// TIA Portal V19 program export: 1 tag tables, 0 data types, 0 data blocks, 5 code blocks (in call order from the OBs), 0 instance data blocks

VAR_GLOBAL   // PLC tag table "Default tag table"
   Stop_All AT %M0.0 : Bool;
   TestTag AT %M0.1 : Bool;
END_VAR

ORGANIZATION_BLOCK "Main"   // OB1, LAD, ProgramCycle
TITLE = "Main Program Sweep (Cycle)"
{ S7_Optimized_Access := 'TRUE' }
// h
// stored: SetENOAutomatically false
   VAR_INPUT
      Initial_Call : Bool;   // Initial call of this OB
      Remanence : Bool;   // =True, if remanent data are available
   END_VAR
   VAR_TEMP
      Start_All : Bool;
      ON : Bool;
   END_VAR
BEGIN

REGION Network 1
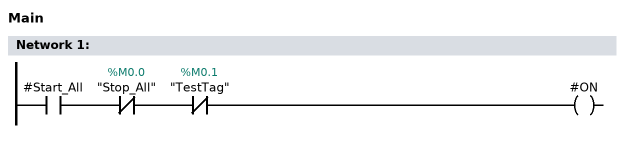
   RUNG wire#powerrail
      Contact( #Start_All )
      I_Contact( "Stop_All" )
      I_Contact( "TestTag" )
      Coil( #ON )
   END_RUNG
   // the same network as SCL:
   #ON := #Start_All AND NOT "Stop_All" AND NOT "TestTag";
END_REGION
END_ORGANIZATION_BLOCK

FUNCTION "NEW_FUNCTION" : Void   // FC2, LAD
TITLE = New Function Added
{ S7_Optimized_Access := 'TRUE' }
// stored: SetENOAutomatically false
BEGIN

REGION Network 1: New Function 1
   // Testing adding a new function.
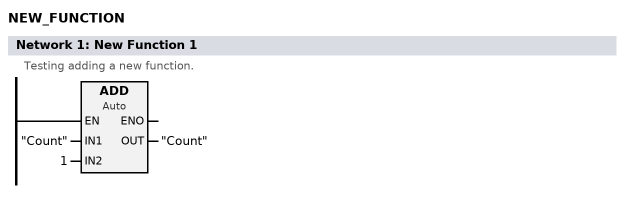
   RUNG wire#powerrail
      Add(in1 := "Count", in2 := 1, out => "Count")
   END_RUNG
   // the same network as SCL:
   "Count" := "Count" + 1;
END_REGION
END_FUNCTION

FUNCTION_BLOCK "SAMPLE_BLOCK"   // FB1, LAD
TITLE = Example Function Block - ie, Multiple Motors Start / Stop
{ S7_Optimized_Access := 'TRUE' }
// stored: MemoryReserve 100, SetENOAutomatically false
BEGIN

REGION Network 1: Drive 1 - Latching
   // Motor 1
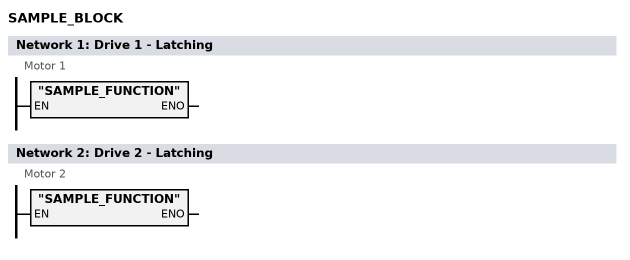
   RUNG wire#powerrail
      "SAMPLE_FUNCTION"()
   END_RUNG
   // the same network as SCL:
   "SAMPLE_FUNCTION"();
END_REGION

REGION Network 2: Drive 2 - Latching
   // Motor 2
   RUNG wire#powerrail
      "SAMPLE_FUNCTION"()
   END_RUNG
   // the same network as SCL:
   "SAMPLE_FUNCTION"();
END_REGION
END_FUNCTION_BLOCK

FUNCTION "SAMPLE_FUNCTION" : Void   // FC1, LAD
TITLE = SAMPLE FUNCTION FOR TESTING DOCUMENTATION
{ S7_Optimized_Access := 'TRUE' }
// stored: SetENOAutomatically false
   VAR_TEMP
      Start : Bool;   // Start Command
      Stop : Bool;   // Stop Command
      Running : Bool;   // Running ? (Y/N)
   END_VAR
BEGIN

REGION Network 1: Basic Latching Function
   // This is A Comment to Test The Documentation Prints Correctly
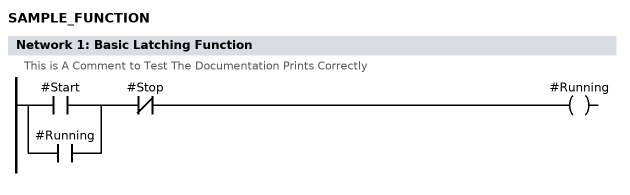
   RUNG wire#powerrail
      Contact( #Start )
      wire#w1
      I_Contact( #Stop )
      Coil( #Running )
   END_RUNG
   RUNG wire#powerrail
      Contact( #Running )
   END_RUNG wire#w1
   // the same network as SCL:
   #Running := (#Start OR #Running) AND NOT #Stop;
END_REGION
END_FUNCTION

FUNCTION_BLOCK "Valve_Example_PWM"   // FB293, LAD
TITLE = Examle Function Block - PWM Valve Control
{ S7_Optimized_Access := 'TRUE' }
// ***For Testing Documentation Only ***
// stored: MemoryReserve 100, SetENOAutomatically false
   VAR_INPUT
      ENable : Bool;
      Rev_Acting : Bool;   // Reverse Acting ( Decrease Output , Valve Closes)
      PV : Real;   // Process Variable
      SP : Real;   // Setpoint
      DB : Real;
      Pulse_TM : Int;
      Pulse_Base : Int;
      Wait_TM : Int;
      Wait_Base : Int;
   END_VAR
   VAR_OUTPUT
      Open_CMD : Bool;
      Close_CMD : Bool;
   END_VAR
   VAR
      Error { ExternalAccessible := 'False'; ExternalVisible := 'False'; ExternalWritable := 'False'} : Real;   // Error Value (Real)
      Abs_Error { ExternalAccessible := 'False'; ExternalVisible := 'False'; ExternalWritable := 'False'} : Real;   // Absolute Error Value
      Neg_Error : Bool;   // Process Variable above Setpoint (eg,Too Low)
      Pos_Error : Bool;   // Process Variable below Setpoint (eg,Too High)
      Open_Reqd : Bool;   // Open Required ( Open Valve Required)
      Close_Reqd : Bool;   // Close Required ( Close Valve Required)
      In_DB : Bool;   // Input Data Block
      Pulse_Time_PT : DInt;
      Pulse_ON_Tmr { S7_SetPoint := 'True'} : TON_TIME;
      Pulse_OFF_Tmr_DN : Bool;
      Pulse_ON_Tmr_DN : Bool;
      Wait_Time_PT : DInt;
      Pulse_OFF_Tmr { S7_SetPoint := 'True'} : TON_TIME;
   END_VAR
   VAR_TEMP
      Pulse_TM_D : DInt;
      Wait_TM_D : DInt;
      DB_LOW_TMP : Real;
   END_VAR
BEGIN

REGION Network 1: Errors
   // Gets error From the Process Variable Minus the Setpoint Value
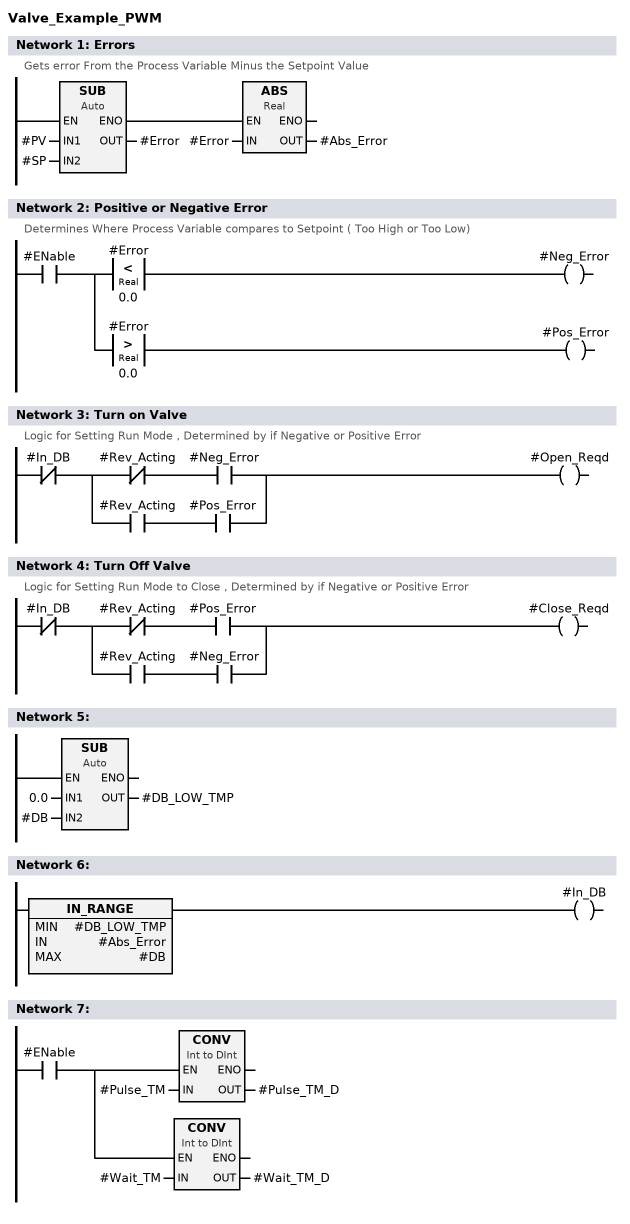
   RUNG wire#powerrail
      Sub(in1 := #PV, in2 := #SP, out => #Error)
      { S7_Templates := "SrcType := Real" } Abs(in := #Error, out => #Abs_Error)
   END_RUNG
   // the same network as SCL:
   #Error := #PV - #SP;
   #Abs_Error := ABS(#Error);
END_REGION

REGION Network 2: Positive or Negative Error
   // Determines Where Process Variable compares to Setpoint ( Too High or Too Low)
   RUNG wire#powerrail
      Contact( #ENable )
      wire#w1
      { S7_Templates := "SrcType := Real" } LT_Contact(in1 := #Error, in2 := 0.0)
      Coil( #Neg_Error )
   END_RUNG
   RUNG wire#w1
      { S7_Templates := "SrcType := Real" } GT_Contact(in1 := #Error, in2 := 0.0)
      Coil( #Pos_Error )
   END_RUNG
   // the same network as SCL:
   #Neg_Error := #ENable AND (#Error < 0.0);
   #Pos_Error := #ENable AND (#Error > 0.0);
END_REGION

REGION Network 3: Turn on Valve
   // Logic for Setting Run Mode , Determined by if Negative or Positive Error
   RUNG wire#powerrail
      I_Contact( #In_DB )
      wire#w1
      I_Contact( #Rev_Acting )
      Contact( #Neg_Error )
      wire#w2
      Coil( #Open_Reqd )
   END_RUNG
   RUNG wire#w1
      Contact( #Rev_Acting )
      Contact( #Pos_Error )
   END_RUNG wire#w2
   // the same network as SCL:
   #Open_Reqd := NOT #In_DB AND ((NOT #Rev_Acting AND #Neg_Error) OR (#Rev_Acting AND #Pos_Error));
END_REGION

REGION Network 4: Turn Off Valve
   // Logic for Setting Run Mode to Close , Determined by if Negative or Positive Error
   RUNG wire#powerrail
      I_Contact( #In_DB )
      wire#w1
      I_Contact( #Rev_Acting )
      Contact( #Pos_Error )
      wire#w2
      Coil( #Close_Reqd )
   END_RUNG
   RUNG wire#w1
      Contact( #Rev_Acting )
      Contact( #Neg_Error )
   END_RUNG wire#w2
   // the same network as SCL:
   #Close_Reqd := NOT #In_DB AND ((NOT #Rev_Acting AND #Pos_Error) OR (#Rev_Acting AND #Neg_Error));
END_REGION

REGION Network 5
   RUNG wire#powerrail
      Sub(in1 := 0.0, in2 := #DB, out => #DB_LOW_TMP)
   END_RUNG
   // the same network as SCL:
   #DB_LOW_TMP := 0.0 - #DB;
END_REGION

REGION Network 6
   RUNG wire#powerrail
      { S7_Templates := "SrcType := Real" } InRange(min := #DB_LOW_TMP, in := #Abs_Error, max := #DB)
      Coil( #In_DB )
   END_RUNG
   // the same network as SCL:
   #In_DB := (#DB_LOW_TMP <= #Abs_Error) AND (#Abs_Error <= #DB);
END_REGION

REGION Network 7
   RUNG wire#powerrail
      Contact( #ENable )
      wire#w1
      { S7_Templates := "[SrcType := Int, DestType := DInt]" } Convert(in := #Pulse_TM, out => #Pulse_TM_D)
   END_RUNG
   RUNG wire#w1
      { S7_Templates := "[SrcType := Int, DestType := DInt]" } Convert(in := #Wait_TM, out => #Wait_TM_D)
   END_RUNG
   // the same network as SCL:
   IF #ENable THEN
       #Pulse_TM_D := INT_TO_DINT(#Pulse_TM);
       #Wait_TM_D := INT_TO_DINT(#Wait_TM);
   END_IF;
END_REGION

REGION Network 8: ***This I just an Example Function and Doesnt Contain all Working netorks *****
END_REGION
END_FUNCTION_BLOCK
